FUNCTION APPEND : STRING(255)
VAR_INPUT
	STRING_TO_APPEND,
	STRING1,
	STRING2:	STRING(255);
END_VAR
VAR
END_VAR

STRING_TO_APPEND := CONCAT(STRING_TO_APPEND, STRING1);
APPEND := CONCAT(STRING_TO_APPEND, STRING2);

END_FUNCTION

(* stored: Version 1.1.0.1, ProductVersion 3.1.4024.9
   POU APPEND: Id {ce0d917d-1e4e-433e-812a-e1ca7a7edc98}, SpecialFunc None *)
